// TwinCAT 3 PLC project mobject_motion
// Title: mobject-motion
// Company: mobject-io-ext
// Author: mobject dev team
// ProjectVersion: 0.0.1
// ProgramVersion: 3.1.4023.0
// libraries:
//   mobject-core, * (mobject.io)
//   Tc2_MC2, * (Beckhoff Automation GmbH)
// project tree:
//   Administrative/ ResetCommand.TcPOU, SetPositionCommand.TcPOU
//   Axis/ Axis.TcPOU, I_Axis.TcIO
//   Base/ AxisCommand.TcPOU, I_AxisCommand.TcIO
//   Homing/ DefaultHomingBuilder.TcPOU, HomingCommand.TcPOU, I_DefaultHomingBuilder.TcIO, I_HomingBuilder.TcIO, I_HomingCommand.TcIO, I_PositioningHomingBuilder.TcIO
//   Moves/ DefaultMoveBuilder.TcPOU, I_JogMoveBuilder.TcIO, I_MoveAbsoluteBuilder.TcIO, I_MoveBuilder.TcIO, I_MoveCommand.TcIO, I_MoveRelativeBuilder.TcIO, MoveAbsoluteCommand.TcPOU, MoveAdditiveCommand.TcPOU, MoveCommand.TcPOU, MoveRelativeCommand.TcPOU, MoveVelocityCommand.TcPOU
//   Stops/ HaltCommand.TcPOU, StopCommand.TcPOU
//   Types/ AxisBufferMode.TcDUT, Direction.TcDUT, EncoderReferenceMode.TcDUT, HomingMode.TcDUT, SetPositionMode.TcDUT

// ---- Types/AxisBufferMode.TcDUT
{attribute 'qualified_only'}
{attribute 'strict'}
TYPE AxisBufferMode :
(
	Aborting := MC_Aborting,
	Buffered := MC_Buffered,
	BlendingLow := MC_BlendingLow,
	BlendingPrevious := MC_BlendingPrevious,
	BlendingNext := MC_BlendingNext,
	BlendingHigh := MC_BlendingHigh
) UINT;
END_TYPE

// ---- Types/Direction.TcDUT
{attribute 'qualified_only'}
{attribute 'strict'}
TYPE Direction :
(
    Position := MC_Positive_Direction,
    ShortestWay := MC_Shortest_Way ,
    Negative := MC_Negative_Direction,
    Current := MC_Current_Direction,
	Undefined := MC_Undefined_Direction
) INT;
END_TYPE

// ---- Types/EncoderReferenceMode.TcDUT
// https://infosys.beckhoff.com/english.php?content=../content/1033/ax5000_system_doku_hw2/649689099.html&id=
{attribute 'qualified_only'}
{attribute 'strict'}
TYPE EncoderReferenceMode :
(
	Default := ENCODERREFERENCEMODE_DEFAULT,
	PLCCam := ENCODERREFERENCEMODE_PLCCAM,
	HardwareSync := ENCODERREFERENCEMODE_HARDWARESYNC,
	HardwareLatchPositive := ENCODERREFERENCEMODE_HARDWARELATCHPOS,
	HardwareLatchNegative := ENCODERREFERENCEMODE_HARDWARELATCHNEG,
	SoftwareSync := ENCODERREFERENCEMODE_SOFTWARESYNC,
	SoftwareLatchPositive := ENCODERREFERENCEMODE_SOFTDRIVELATCHPOS,
	SoftwareLatchNegative := ENCODERREFERENCEMODE_SOFTDRIVELATCHNEG
) UDINT;
END_TYPE

// ---- Types/HomingMode.TcDUT
{attribute 'qualified_only'}
{attribute 'strict'}
TYPE HomingMode :
(
	Default := MC_DefaultHoming,
	Direct := MC_Direct,
	ForceCalibration := MC_ForceCalibration,
	ResetCalibration := MC_ResetCalibration
) INT;
END_TYPE

// ---- Types/SetPositionMode.TcDUT
{attribute 'qualified_only'}
{attribute 'strict'}
TYPE SetPositionMode :
(
	Absolute,
	Relative
);
END_TYPE

// ---- Axis/I_Axis.TcIO
INTERFACE I_Axis

PROPERTY INTERNAL _InternalAxisRef : REFERENCE TO Tc2_MC2.AXIS_REF
GET
END_GET
END_PROPERTY

PROPERTY INTERNAL _InternalJog : REFERENCE TO MC_Jog
GET
END_GET
END_PROPERTY

PROPERTY INTERNAL _InternalParameterSet : REFERENCE TO ST_AxisParameterSet
GET
END_GET
END_PROPERTY

PROPERTY AxisId : UDINT
GET
END_GET
END_PROPERTY

{warning 'add property implementation'}
PROPERTY BufferMode : Tc2_MC2.MC_BufferMode
GET
END_GET
SET
END_SET
END_PROPERTY

PROPERTY Busy : BOOL
GET
END_GET
END_PROPERTY

METHOD Disable
END_METHOD

METHOD DisableNegative
END_METHOD

METHOD DisablePositive
END_METHOD

METHOD Enable
VAR_INPUT
	bufferMode : AxisBufferMode;
END_VAR
END_METHOD

METHOD EnableNegative : BOOL
END_METHOD

METHOD EnablePositive
END_METHOD

PROPERTY ErrorId : UDINT
GET
END_GET
END_PROPERTY

METHOD Halt
VAR_INPUT
	feedback : REFERENCE TO I_CommandFeedback;
END_VAR
END_METHOD

PROPERTY HasError : BOOL
GET
END_GET
END_PROPERTY

METHOD HomingBuilder : I_HomingBuilder
END_METHOD

PROPERTY IsAccelerating : BOOL
GET
END_GET
END_PROPERTY

PROPERTY IsAtConstantVelocity : BOOL
GET
END_GET
END_PROPERTY

PROPERTY IsAtStandStill : BOOL
GET
END_GET
END_PROPERTY

PROPERTY IsDecelerating : BOOL
GET
END_GET
END_PROPERTY

PROPERTY IsErrorStopped : BOOL
GET
END_GET
END_PROPERTY

PROPERTY IsHoming : BOOL
GET
END_GET
END_PROPERTY

PROPERTY IsInContinuousMotion : BOOL
GET
END_GET
END_PROPERTY

PROPERTY IsInDiscreteMotion : BOOL
GET
END_GET
END_PROPERTY

PROPERTY IsInSynchronizedMotion : BOOL
GET
END_GET
END_PROPERTY

PROPERTY IsReady : BOOL
GET
END_GET
END_PROPERTY

PROPERTY IsStatusValid : BOOL
GET
END_GET
END_PROPERTY

PROPERTY IsStopping : BOOL
GET
END_GET
END_PROPERTY

METHOD JogBackwards
VAR_INPUT
	velocity : LREAL;
END_VAR
END_METHOD

METHOD JogForward
VAR_INPUT
	velocity : LREAL;
END_VAR
END_METHOD

METHOD MoveBuilder : I_MoveBuilder
END_METHOD

PROPERTY Override : LREAL
GET
END_GET
SET
END_SET
END_PROPERTY

METHOD Reset
VAR_INPUT
	feedback : REFERENCE TO I_CommandFeedback;
END_VAR
END_METHOD

METHOD SetPositionAbsolute
VAR_INPUT
	positionToSet : LREAL;
	feedback : REFERENCE TO I_CommandFeedback;
END_VAR
END_METHOD

METHOD SetPositionRelative
VAR_INPUT
	distanceToShift : LREAL;
	feedback : REFERENCE TO I_CommandFeedback;
END_VAR
END_METHOD

METHOD Stop
VAR_INPUT
	feedback : REFERENCE TO I_CommandFeedback;
END_VAR
END_METHOD

METHOD StopJogging
END_METHOD

END_INTERFACE

// ---- Base/I_AxisCommand.TcIO
INTERFACE I_AxisCommand EXTENDS I_Command

END_INTERFACE

// ---- Homing/I_DefaultHomingBuilder.TcIO
INTERFACE I_DefaultHomingBuilder EXTENDS __System.IQueryInterface

METHOD BuildDefaultHomingCommand : I_HomingCommand
END_METHOD

METHOD Cam : I_DefaultHomingBuilder
VAR_INPUT
	value : REFERENCE TO BOOL;
END_VAR
END_METHOD

METHOD ClearLag : I_PositioningHomingBuilder
END_METHOD

METHOD KeepLag : I_PositioningHomingBuilder
END_METHOD

METHOD Position : I_PositioningHomingBuilder
VAR_INPUT
	value : LREAL;
END_VAR
END_METHOD

METHOD ReferenceMode : I_DefaultHomingBuilder
VAR_INPUT
	value : EncoderReferenceMode;
END_VAR
END_METHOD

METHOD SearchDirection : I_DefaultHomingBuilder
VAR_INPUT
	value : Direction;
END_VAR
END_METHOD

METHOD SearchVelocity : I_DefaultHomingBuilder
VAR_INPUT
	value : LREAL;
END_VAR
END_METHOD

METHOD SyncDirection : I_DefaultHomingBuilder
VAR_INPUT
	value : Direction;
END_VAR
END_METHOD

METHOD SyncVelocity : I_DefaultHomingBuilder
VAR_INPUT
	value : LREAL;
END_VAR
END_METHOD

END_INTERFACE

// ---- Homing/I_HomingBuilder.TcIO
INTERFACE I_HomingBuilder EXTENDS __System.IQueryInterface

METHOD BuildForceCalibrationCommand : I_HomingCommand
END_METHOD

METHOD BuildResetCalibrationCommand : I_HomingCommand
END_METHOD

METHOD Position : I_PositioningHomingBuilder
VAR_INPUT
	value : LREAL;
END_VAR
END_METHOD

END_INTERFACE

// ---- Homing/I_HomingCommand.TcIO
INTERFACE I_HomingCommand EXTENDS I_AxisCommand

END_INTERFACE

// ---- Homing/I_PositioningHomingBuilder.TcIO
INTERFACE I_PositioningHomingBuilder EXTENDS __System.IQueryInterface

METHOD BuildDefaultHomingCommand : I_HomingCommand
END_METHOD

METHOD BuildDirectHomingCommand : I_HomingCommand
END_METHOD

METHOD Cam : I_DefaultHomingBuilder
VAR_INPUT
	value : REFERENCE TO BOOL;
END_VAR
END_METHOD

METHOD ClearLag : I_PositioningHomingBuilder
END_METHOD

METHOD KeepLag : I_PositioningHomingBuilder
END_METHOD

METHOD Position : I_PositioningHomingBuilder
VAR_INPUT
	value : LREAL;
END_VAR
END_METHOD

METHOD ReferenceMode : I_DefaultHomingBuilder
VAR_INPUT
	value : EncoderReferenceMode;
END_VAR
END_METHOD

METHOD SearchDirection : I_DefaultHomingBuilder
VAR_INPUT
	value : Direction;
END_VAR
END_METHOD

METHOD SearchVelocity : I_DefaultHomingBuilder
VAR_INPUT
	value : LREAL;
END_VAR
END_METHOD

METHOD SyncDirection : I_DefaultHomingBuilder
VAR_INPUT
	value : Direction;
END_VAR
END_METHOD

METHOD SyncVelocity : I_DefaultHomingBuilder
VAR_INPUT
	value : LREAL;
END_VAR
END_METHOD

END_INTERFACE

// ---- Moves/I_JogMoveBuilder.TcIO
INTERFACE I_JogMoveBuilder EXTENDS __System.IQueryInterface

METHOD Acceleration : I_MoveBuilder
VAR_INPUT
	value : LREAL;
END_VAR
END_METHOD

METHOD BuildBackwardsCommand : I_MoveCommand
END_METHOD

METHOD BuildForwardCommand : I_MoveCommand
END_METHOD

METHOD Deceleration : I_MoveBuilder
VAR_INPUT
	value : LREAL;
END_VAR
END_METHOD

METHOD Distance : I_JogMoveBuilder
VAR_INPUT
	value : LREAL;
END_VAR
END_METHOD

METHOD Jerk : I_MoveBuilder
VAR_INPUT
	value : LREAL;
END_VAR
END_METHOD

METHOD Velocity : I_MoveBuilder
VAR_INPUT
	value : LREAL;
END_VAR
END_METHOD

END_INTERFACE

// ---- Moves/I_MoveAbsoluteBuilder.TcIO
INTERFACE I_MoveAbsoluteBuilder EXTENDS __System.IQueryInterface

METHOD Acceleration : I_MoveBuilder
VAR_INPUT
	value : LREAL;
END_VAR
END_METHOD

METHOD BufferMode : I_MoveBuilder
VAR_INPUT
	mode : AxisBufferMode;
END_VAR
END_METHOD

METHOD BuildMoveAbsoluteCommand : I_MoveCommand
END_METHOD

METHOD Deceleration : I_MoveBuilder
VAR_INPUT
	value : LREAL;
END_VAR
END_METHOD

METHOD Jerk : I_MoveBuilder
VAR_INPUT
	value : LREAL;
END_VAR
END_METHOD

METHOD Position : I_MoveAbsoluteBuilder
VAR_INPUT
	value : LREAL;
END_VAR
END_METHOD

METHOD Velocity : I_MoveBuilder
VAR_INPUT
	value : LREAL;
END_VAR
END_METHOD

END_INTERFACE

// ---- Moves/I_MoveBuilder.TcIO
INTERFACE I_MoveBuilder EXTENDS __System.IQueryInterface

METHOD Acceleration : I_MoveBuilder
VAR_INPUT
	value : LREAL;
END_VAR
END_METHOD

METHOD BufferMode : I_MoveBuilder
VAR_INPUT
	mode : AxisBufferMode;
END_VAR
END_METHOD

METHOD BuildMoveVelocityCommand : I_MoveCommand
END_METHOD

METHOD Deceleration : I_MoveBuilder
VAR_INPUT
	value : LREAL;
END_VAR
END_METHOD

METHOD Distance : I_MoveRelativeBuilder
VAR_INPUT
	value : LREAL;
END_VAR
END_METHOD

METHOD Jerk : I_MoveBuilder
VAR_INPUT
	value : LREAL;
END_VAR
END_METHOD

METHOD Position : I_MoveAbsoluteBuilder
VAR_INPUT
	value : LREAL;
END_VAR
END_METHOD

METHOD Velocity : I_MoveBuilder
VAR_INPUT
	value : LREAL;
END_VAR
END_METHOD

END_INTERFACE

// ---- Moves/I_MoveCommand.TcIO
INTERFACE I_MoveCommand EXTENDS I_Command

END_INTERFACE

// ---- Moves/I_MoveRelativeBuilder.TcIO
INTERFACE I_MoveRelativeBuilder EXTENDS __System.IQueryInterface

METHOD Acceleration : I_MoveBuilder
VAR_INPUT
	value : LREAL;
END_VAR
END_METHOD

METHOD BufferMode : I_MoveBuilder
VAR_INPUT
	mode : AxisBufferMode;
END_VAR
END_METHOD

METHOD BuildMoveAdditiveCommand : I_MoveCommand
END_METHOD

METHOD BuildMoveRelativeCommand : I_MoveCommand
END_METHOD

METHOD Deceleration : I_MoveBuilder
VAR_INPUT
	value : LREAL;
END_VAR
END_METHOD

METHOD Distance : I_MoveRelativeBuilder
VAR_INPUT
	value : LREAL;
END_VAR
END_METHOD

METHOD Jerk : I_MoveBuilder
VAR_INPUT
	value : LREAL;
END_VAR
END_METHOD

METHOD Velocity : I_MoveBuilder
VAR_INPUT
	value : LREAL;
END_VAR
END_METHOD

END_INTERFACE

// ---- Administrative/ResetCommand.TcPOU
{attribute 'linkalways'} 
{attribute 'no_explicit_call' := 'This FB is a CLASS and must be accessed using methods or properties'}
{attribute 'enable_dynamic_creation'}
FUNCTION_BLOCK ResetCommand EXTENDS AxisCommand

METHOD FB_init : BOOL
VAR_INPUT
	bInitRetains : BOOL; // if TRUE, the retain variables are initialized (warm start / cold start)
	bInCopyCode : BOOL;  // if TRUE, the instance afterwards gets moved into the copy code (online change)
	axis : I_Axis;
END_VAR
_axis := axis;
END_METHOD

METHOD PROTECTED  WhileBusy
VAR_INPUT
	CommandState : I_CommandBusyState;
END_VAR
VAR_INST
	_fb : MC_Reset;
END_VAR
_fb(
	Axis := _axis._InternalAxisRef,
	Execute := TRUE
);

IF _fb.Busy THEN
	RETURN;
END_IF

_fb(Axis := _axis._InternalAxisRef, Execute := FALSE);

IF _fb.Error THEN
	CommandState.SetError(_fb.ErrorID);
	RETURN;
END_IF

CommandState.SetDone();
END_METHOD

END_FUNCTION_BLOCK

// ---- Base/AxisCommand.TcPOU
{attribute 'linkalways'} 
{attribute 'no_explicit_call' := 'This FB is a CLASS and must be accessed using methods or properties'}
{attribute 'enable_dynamic_creation'}
FUNCTION_BLOCK ABSTRACT AxisCommand EXTENDS Command IMPLEMENTS I_AxisCommand
VAR
	_axis : I_Axis;
END_VAR

END_FUNCTION_BLOCK

// ---- Axis/Axis.TcPOU
{attribute 'linkalways'} 
{attribute 'no_explicit_call' := 'This FB is a CLASS and must be accessed using methods or properties'}
{attribute 'enable_dynamic_creation'}
FUNCTION_BLOCK Axis EXTENDS CyclicInstance IMPLEMENTS I_Axis
VAR
	_axisRef : Tc2_MC2.AXIS_REF;
	_power : MC_Power;
	_jog : MC_Jog;
	_readStatus : MC_ReadStatus;
	_parameterSet : ST_AxisParameterSet;
	
	_enable : BOOL;
	_enablePositive : BOOL;
	_enableNegative : BOOL;
	
	_override : LREAL := 100.0;
	_powerBufferMode : AxisBufferMode := AxisBufferMode.Aborting;
END_VAR

PROPERTY PUBLIC _InternalAxisRef : REFERENCE TO Tc2_MC2.AXIS_REF
GET
_InternalAxisRef REF= _axisRef;
END_GET
END_PROPERTY

PROPERTY PUBLIC _InternalJog : REFERENCE TO MC_Jog
GET
_InternalJog REF= _jog;
END_GET
END_PROPERTY

PROPERTY PUBLIC _InternalParameterSet : REFERENCE TO ST_AxisParameterSet
GET
_InternalParameterSet REF= _parameterSet;
END_GET
END_PROPERTY

PROPERTY AxisId : UDINT
GET
AxisId := _axisRef.NcToPlc.AxisId;
END_GET
END_PROPERTY

{warning 'add property implementation'}
PROPERTY BufferMode : Tc2_MC2.MC_BufferMode
GET
END_GET
SET
END_SET
END_PROPERTY

PROPERTY Busy : BOOL
GET
END_GET
END_PROPERTY

METHOD  CyclicCall
VAR_INST
	_readParameterSet : MC_ReadParameterSet;
	parameterSetRead : BOOL;
END_VAR
_power(
	Axis := THIS^._axisRef,
	Enable := THIS^._enable,
	Enable_Positive := THIS^._enablePositive,
	Enable_Negative := THIS^._enableNegative,
	Override := THIS^._override,
	BufferMode := THIS^._powerBufferMode
);

_readStatus(
	Axis := THIS^._axisRef,
	Enable := _enable
);

IF NOT parameterSetRead THEN
	_readParameterSet(
		Axis := THIS^._axisRef,
		Parameter := _parameterSet,
		Execute := TRUE
	);
	
	IF NOT _readParameterSet.Busy THEN
		_readParameterSet(
			Axis := THIS^._axisRef,
			Parameter := _parameterSet,
			Execute := TRUE
		);
		IF _readParameterSet.Done THEN
			parameterSetRead := TRUE;
		END_IF
	END_IF
END_IF
END_METHOD

METHOD Disable
_enable := FALSE;
END_METHOD

METHOD DisableNegative
_enableNegative := FALSE;
END_METHOD

METHOD DisablePositive
_enablePositive := FALSE;
END_METHOD

METHOD Enable
VAR_INPUT
	bufferMode : AxisBufferMode;
END_VAR
_enable := TRUE;
_powerBufferMode := bufferMode;
END_METHOD

METHOD EnableNegative : BOOL
_enableNegative := TRUE;
END_METHOD

METHOD EnablePositive
_enablePositive := TRUE;
END_METHOD

PROPERTY ErrorId : UDINT
GET
ErrorId := _readStatus.ErrorID;
END_GET
END_PROPERTY

METHOD Halt
VAR_INPUT
	feedback : REFERENCE TO I_CommandFeedback;
END_VAR
VAR_INST
	pCmd : POINTER TO HaltCommand;
END_VAR
pCmd := __NEW(HaltCommand(axis := THIS^));
pCmd^.Execute(feedback).ThenRelease();
END_METHOD

PROPERTY HasError : BOOL
GET
HasError := _readStatus.Error;
END_GET
END_PROPERTY

METHOD HomingBuilder : I_HomingBuilder
VAR_INST
	builder : DefaultHomingBuilder(axis := THIS^);
END_VAR
HomingBuilder := builder;
END_METHOD

PROPERTY IsAccelerating : BOOL
GET
IsAccelerating := _readStatus.Accelerating;
END_GET
END_PROPERTY

PROPERTY IsAtConstantVelocity : BOOL
GET
IsAtConstantVelocity := _readStatus.ConstantVelocity;
END_GET
END_PROPERTY

PROPERTY IsAtStandStill : BOOL
GET
IsAtStandStill := _readStatus.StandStill;
END_GET
END_PROPERTY

PROPERTY IsDecelerating : BOOL
GET
IsDecelerating := _readStatus.Decelerating;
END_GET
END_PROPERTY

PROPERTY IsErrorStopped : BOOL
GET
IsErrorStopped := _readStatus.ErrorStop;
END_GET
END_PROPERTY

PROPERTY IsHoming : BOOL
GET
IsHoming := _readStatus.Homing;
END_GET
END_PROPERTY

PROPERTY IsInContinuousMotion : BOOL
GET
IsInContinuousMotion := _readStatus.ContinuousMotion;
END_GET
END_PROPERTY

PROPERTY IsInDiscreteMotion : BOOL
GET
IsInDiscreteMotion := _readStatus.DiscreteMotion;
END_GET
END_PROPERTY

PROPERTY IsInSynchronizedMotion : BOOL
GET
IsInSynchronizedMotion := _readStatus.SynchronizedMotion;
END_GET
END_PROPERTY

PROPERTY IsReady : BOOL
GET
IsReady := _power.Status;
END_GET
END_PROPERTY

PROPERTY IsStatusValid : BOOL
GET
IsStatusValid := _readStatus.Valid;
END_GET
END_PROPERTY

PROPERTY IsStopping : BOOL
GET
IsStopping := _readStatus.Stopping;
END_GET
END_PROPERTY

METHOD JogBackwards
VAR_INPUT
	velocity : LREAL;
END_VAR
_jog(
	Axis := _axisRef,
	JogForward := FALSE,
	JogBackwards := TRUE,
	Mode := MC_JOGMODE_CONTINOUS,
	Velocity := velocity
);
END_METHOD

METHOD JogForward
VAR_INPUT
	velocity : LREAL;
END_VAR
_jog(
	Axis := _axisRef,
	JogForward := TRUE,
	JogBackwards := FALSE,
	Mode := MC_JOGMODE_CONTINOUS,
	Velocity := velocity
);
END_METHOD

METHOD MoveBuilder : I_MoveBuilder
VAR_INST
	builder : DefaultMoveBuilder(axis := THIS^);
END_VAR
MoveBuilder := builder;
END_METHOD

PROPERTY Override : LREAL
GET
Override := _override;
END_GET
SET
_override := Override;
END_SET
END_PROPERTY

METHOD Reset
VAR_INPUT
	feedback : REFERENCE TO I_CommandFeedback;
END_VAR
VAR_INST
	pCmd : POINTER TO ResetCommand;
END_VAR
pCmd := __NEW(ResetCommand(axis := THIS^));
pCmd^.Execute(feedback).ThenRelease();
END_METHOD

METHOD SetPositionAbsolute
VAR_INPUT
	positionToSet : LREAL;
	feedback : REFERENCE TO I_CommandFeedback;
END_VAR
VAR_INST
	pCmd : POINTER TO SetPositionCommand;
END_VAR
pCmd := __NEW(SetPositionCommand(axis := THIS^, position := positionToSet, mode := SetPositionMode.Absolute));
pCmd^.Execute(feedback).ThenRelease();
END_METHOD

METHOD SetPositionRelative
VAR_INPUT
	distanceToShift : LREAL;
	feedback : REFERENCE TO I_CommandFeedback;
END_VAR
VAR_INST
	pCmd : POINTER TO SetPositionCommand;
END_VAR
pCmd := __NEW(SetPositionCommand(axis := THIS^, position := distanceToShift, mode := SetPositionMode.Relative));
pCmd^.Execute(feedback).ThenRelease();
END_METHOD

METHOD Stop
VAR_INPUT
	feedback : REFERENCE TO I_CommandFeedback;
END_VAR
VAR_INST
	pCmd : POINTER TO StopCommand;
END_VAR
pCmd := __NEW(StopCommand(axis := THIS^));
pCmd^.Execute(feedback).ThenRelease();
END_METHOD

METHOD StopJogging
_jog(
	Axis := _axisRef,
	JogForward := FALSE,
	JogBackwards := FALSE,
);
END_METHOD

END_FUNCTION_BLOCK

// ---- Stops/HaltCommand.TcPOU
{attribute 'linkalways'} 
{attribute 'no_explicit_call' := 'This FB is a CLASS and must be accessed using methods or properties'}
{attribute 'enable_dynamic_creation'}
FUNCTION_BLOCK HaltCommand EXTENDS AxisCommand
VAR
	_deceleration : LREAL;
	_jerk : LREAL;
	_bufferMode : AxisBufferMode;
END_VAR

METHOD FB_init : BOOL
VAR_INPUT
	bInitRetains : BOOL; // if TRUE, the retain variables are initialized (warm start / cold start)
	bInCopyCode : BOOL;  // if TRUE, the instance afterwards gets moved into the copy code (online change)
	axis : I_Axis;
END_VAR
_axis := axis;
END_METHOD

METHOD PROTECTED  WhileBusy
VAR_INPUT
	CommandState : I_CommandBusyState;
END_VAR
VAR_INST
	_fb : MC_Halt;
END_VAR
_fb(
	Axis := _axis._InternalAxisRef,
	Execute := TRUE,
	Deceleration := _deceleration,
	Jerk := _jerk,
	BufferMode := _bufferMode
);

IF _fb.Busy THEN
	RETURN;
END_IF

_fb(Axis := _axis._InternalAxisRef, Execute := FALSE);

IF _fb.CommandAborted THEN
	CommandState.SetAborting();
	RETURN;
END_IF

IF _fb.Error THEN
	CommandState.SetError(_fb.ErrorID);
	RETURN;
END_IF

CommandState.SetDone();
END_METHOD

END_FUNCTION_BLOCK

// ---- Homing/DefaultHomingBuilder.TcPOU
{attribute 'linkalways'} 
{attribute 'no_explicit_call' := 'This FB is a CLASS and must be accessed using methods or properties'}
{attribute 'enable_dynamic_creation'}
FUNCTION_BLOCK DefaultHomingBuilder IMPLEMENTS I_HomingBuilder, I_PositioningHomingBuilder, I_DefaultHomingBuilder
VAR
	_axis : I_Axis;
	_position : LREAL;
	_options : ST_HomingOptions;
	_cam : REFERENCE TO BOOL;
END_VAR

METHOD BuildDefaultHomingCommand : I_HomingCommand
VAR
	pCmd : POINTER TO HomingCommand;
	cmd : I_HomingCommand;
END_VAR
pCmd := __NEW(HomingCommand(
	axis := _axis,
	position := _position,
	mode := HomingMode.Default,
	options := _options,
	cam := _cam
));
BuildDefaultHomingCommand := pCmd^;
END_METHOD

METHOD BuildDirectHomingCommand : I_HomingCommand
VAR
	pCmd : POINTER TO HomingCommand;
	cmd : I_HomingCommand;
	null : BOOL;
END_VAR
pCmd := __NEW(HomingCommand(
	axis := _axis,
	position := _position,
	mode := HomingMode.Direct,
	options := _options,
	cam := null
));
BuildDirectHomingCommand := pCmd^;
END_METHOD

METHOD BuildForceCalibrationCommand : I_HomingCommand
VAR
	pCmd : POINTER TO HomingCommand;
	cmd : I_HomingCommand;
	null : BOOL;
END_VAR
pCmd := __NEW(HomingCommand(
	axis := _axis,
	position := _position,
	mode := HomingMode.ForceCalibration,
	options := _options,
	cam := null
));
BuildForceCalibrationCommand := pCmd^;
END_METHOD

METHOD BuildResetCalibrationCommand : I_HomingCommand
VAR
	pCmd : POINTER TO HomingCommand;
	cmd : I_HomingCommand;
	null : BOOL;
END_VAR
pCmd := __NEW(HomingCommand(
	axis := _axis,
	position := _position,
	mode := HomingMode.ResetCalibration,
	options := _options,
	cam := null
));
BuildResetCalibrationCommand := pCmd^;
END_METHOD

METHOD Cam : I_DefaultHomingBuilder
VAR_INPUT
	value : REFERENCE TO BOOL;
END_VAR
_cam REF= value;
Cam := THIS^;
END_METHOD

METHOD ClearLag : I_PositioningHomingBuilder
_options.ClearPositionLag := TRUE;
ClearLag := THIS^;
END_METHOD

METHOD FB_init : BOOL
VAR_INPUT
	bInitRetains : BOOL; // if TRUE, the retain variables are initialized (warm start / cold start)
	bInCopyCode : BOOL;  // if TRUE, the instance afterwards gets moved into the copy code (online change)
	axis : I_Axis;
END_VAR
_axis := axis;
END_METHOD

METHOD KeepLag : I_PositioningHomingBuilder
_options.ClearPositionLag := FALSE;
KeepLag := THIS^;
END_METHOD

METHOD Position : I_PositioningHomingBuilder
VAR_INPUT
	value : LREAL;
END_VAR
_position := value;
Position := THIS^;
END_METHOD

METHOD ReferenceMode : I_DefaultHomingBuilder
VAR_INPUT
	value : EncoderReferenceMode;
END_VAR
_options.ReferenceMode := value;
ReferenceMode := THIS^;
END_METHOD

METHOD SearchDirection : I_DefaultHomingBuilder
VAR_INPUT
	value : Direction;
END_VAR
_options.SearchDirection := value;
SearchDirection := THIS^;
END_METHOD

METHOD SearchVelocity : I_DefaultHomingBuilder
VAR_INPUT
	value	: LREAL;
END_VAR
_options.SearchVelocity := value;
SearchVelocity := THIS^;
END_METHOD

METHOD SyncDirection : I_DefaultHomingBuilder
VAR_INPUT
	value : Direction;
END_VAR
_options.SyncDirection := value;
SyncDirection := THIS^;
END_METHOD

METHOD SyncVelocity : I_DefaultHomingBuilder
VAR_INPUT
	value : LREAL;
END_VAR
_options.SyncVelocity := value;
SyncVelocity := THIS^;
END_METHOD

END_FUNCTION_BLOCK

// ---- Homing/HomingCommand.TcPOU
{attribute 'linkalways'} 
{attribute 'no_explicit_call' := 'This FB is a CLASS and must be accessed using methods or properties'}
{attribute 'enable_dynamic_creation'}
FUNCTION_BLOCK HomingCommand EXTENDS AxisCommand IMPLEMENTS I_HomingCommand
VAR
	_fb : MC_Home;
	_position : LREAL;
	_mode : HomingMode;
	_options : ST_HomingOptions;
	_cam : REFERENCE TO BOOL;
END_VAR

METHOD FB_init : BOOL
VAR_INPUT
	bInitRetains : BOOL; // if TRUE, the retain variables are initialized (warm start / cold start)
	bInCopyCode : BOOL;  // if TRUE, the instance afterwards gets moved into the copy code (online change)
	axis : I_Axis;
	position : LREAL;
	mode : HomingMode;
	options : ST_HomingOptions;
	cam : REFERENCE TO BOOL;
END_VAR
_axis := axis;
_position := position;
_mode := mode;
_options := options;
IF __ISVALIDREF(cam) THEN
	_cam REF= cam;
END_IF
END_METHOD

METHOD PROTECTED  WhileBusy
VAR_INPUT
	CommandState : I_CommandBusyState;
END_VAR
VAR
	_dummy : BOOL := FALSE;
END_VAR
VAR_INST
	_fb : MC_Home;
END_VAR
IF NOT __ISVALIDREF(_cam) THEN
	_cam REF= _dummy;
END_IF

_fb(
	Axis := _axis._InternalAxisRef,
	Execute := TRUE,
	Position := _position,
	HomingMode := _mode,
	Options := _options,
	bCalibrationCam := _cam
);

IF _fb.Busy THEN
	RETURN;
END_IF

IF _fb.CommandAborted THEN
	_fb(Axis := _axis._InternalAxisRef, Execute := FALSE);
	CommandState.SetAborting();
	RETURN;
END_IF

IF _fb.Error THEN
	_fb(Axis := _axis._InternalAxisRef, Execute := FALSE);
	CommandState.SetError(_fb.ErrorID);
	RETURN;
END_IF

_fb(Axis := _axis._InternalAxisRef, Execute := FALSE);
CommandState.SetDone();
END_METHOD

END_FUNCTION_BLOCK

// ---- Moves/DefaultMoveBuilder.TcPOU
{attribute 'linkalways'} 
{attribute 'no_explicit_call' := 'This FB is a CLASS and must be accessed using methods or properties'}
{attribute 'enable_dynamic_creation'}
FUNCTION_BLOCK DefaultMoveBuilder IMPLEMENTS I_MoveBuilder, I_MoveAbsoluteBuilder, I_MoveRelativeBuilder
VAR
	_axis : I_Axis;
	_position : LREAL;
	_distance : LREAL;
	_velocity : LREAL;
	_acceleration: LREAL;
	_deceleration: LREAL;
	_jerk: LREAL;
	_bufferMode: AxisBufferMode;
END_VAR

METHOD Acceleration : I_MoveBuilder
VAR_INPUT
	value : LREAL;
END_VAR
_acceleration := value;
Acceleration := THIS^;
END_METHOD

METHOD BufferMode : I_MoveBuilder
VAR_INPUT
	mode : AxisBufferMode;
END_VAR
_bufferMode := mode;
BufferMode := THIS^;
END_METHOD

METHOD BuildMoveAbsoluteCommand : I_MoveCommand
VAR
	pCmd : POINTER TO MoveAbsoluteCommand;
	cmd : I_MoveCommand;
END_VAR
pCmd := __NEW(MoveAbsoluteCommand(
	axis := _axis,
	position := _position,
	velocity := _velocity,
	acceleration := _acceleration,
	deceleration := _deceleration,
	jerk := _jerk,
	bufferMode := _bufferMode
));
BuildMoveAbsoluteCommand := pCmd^;
END_METHOD

METHOD BuildMoveAdditiveCommand : I_MoveCommand
VAR
	pCmd : POINTER TO MoveAdditiveCommand;
	cmd : I_MoveCommand;
END_VAR
pCmd := __NEW(MoveAdditiveCommand(
	axis := _axis,
	distance := _distance,
	velocity := _velocity,
	acceleration := _acceleration,
	deceleration := _deceleration,
	jerk := _jerk,
	bufferMode := _bufferMode
));
BuildMoveAdditiveCommand := pCmd^;
END_METHOD

METHOD BuildMoveRelativeCommand : I_MoveCommand
VAR
	pCmd : POINTER TO MoveRelativeCommand;
	cmd : I_MoveCommand;
END_VAR
pCmd := __NEW(MoveRelativeCommand(
	axis := _axis,
	distance := _distance,
	velocity := _velocity,
	acceleration := _acceleration,
	deceleration := _deceleration,
	jerk := _jerk,
	bufferMode := _bufferMode
));
BuildMoveRelativeCommand := pCmd^;
END_METHOD

METHOD BuildMoveVelocityCommand : I_MoveCommand
VAR
	pCmd : POINTER TO MoveVelocityCommand;
	cmd : I_MoveCommand;
END_VAR
pCmd := __NEW(MoveVelocityCommand(
	axis := _axis,
	velocity := _velocity,
	acceleration := _acceleration,
	deceleration := _deceleration,
	jerk := _jerk,
	bufferMode := _bufferMode
));
BuildMoveVelocityCommand := pCmd^;
END_METHOD

METHOD Deceleration : I_MoveBuilder
VAR_INPUT
	value : LREAL;
END_VAR
_deceleration := value;
Deceleration := THIS^;
END_METHOD

METHOD Distance : I_MoveRelativeBuilder
VAR_INPUT
	value : LREAL;
END_VAR
_distance := value;
Distance := THIS^;
END_METHOD

METHOD FB_init : BOOL
VAR_INPUT
	bInitRetains : BOOL; // if TRUE, the retain variables are initialized (warm start / cold start)
	bInCopyCode : BOOL;  // if TRUE, the instance afterwards gets moved into the copy code (online change)
	axis : I_Axis;
END_VAR
_axis := axis;
END_METHOD

METHOD Jerk : I_MoveBuilder
VAR_INPUT
	value : LREAL;
END_VAR
_jerk := value;
Jerk := THIS^;
END_METHOD

METHOD Position : I_MoveAbsoluteBuilder
VAR_INPUT
	value : LREAL;
END_VAR
_position := value;
Position := THIS^;
END_METHOD

METHOD Velocity : I_MoveBuilder
VAR_INPUT
	value : LREAL;
END_VAR
IF value <= 0 THEN
	_velocity := _axis._InternalParameterSet.fDriveVeloReferenz;
ELSE
	_velocity := value;
END_IF
Velocity := THIS^;
END_METHOD

END_FUNCTION_BLOCK

// ---- Moves/MoveAbsoluteCommand.TcPOU
{attribute 'linkalways'} 
{attribute 'no_explicit_call' := 'This FB is a CLASS and must be accessed using methods or properties'}
{attribute 'enable_dynamic_creation'}
FUNCTION_BLOCK INTERNAL MoveAbsoluteCommand EXTENDS MoveCommand
VAR
	_fb : MC_MoveAbsolute;
	_position : LREAL;
END_VAR

METHOD FB_init : BOOL
VAR_INPUT
	bInitRetains : BOOL; // if TRUE, the retain variables are initialized (warm start / cold start)
	bInCopyCode : BOOL;  // if TRUE, the instance afterwards gets moved into the copy code (online change)
	axis : I_Axis;
	position : LREAL;
	velocity : LREAL;
	acceleration : LREAL;
	deceleration : LREAL;
	jerk : LREAL;
	bufferMode : AxisBufferMode;
END_VAR
_axis := axis;
_position := position;
_velocity := velocity;
_acceleration := acceleration;
_deceleration := deceleration;
_jerk := jerk;
_bufferMode := bufferMode;
END_METHOD

METHOD PROTECTED WhileBusy
VAR_INPUT
	CommandState : I_CommandBusyState;
END_VAR
_fb(
	Axis := _axis._InternalAxisRef,
	Execute := TRUE,
	Position := _position,
	Velocity := _velocity,
	Acceleration := _acceleration,
	Deceleration := _deceleration,
	Jerk := _jerk,
	BufferMode := _bufferMode
);

IF _fb.Busy THEN
	RETURN;
END_IF

IF _fb.CommandAborted THEN
	_fb(Axis := _axis._InternalAxisRef, Execute := FALSE);
	CommandState.SetAborting();
	RETURN;
END_IF

IF _fb.Error THEN
	_fb(Axis := _axis._InternalAxisRef, Execute := FALSE);
	CommandState.SetError(_fb.ErrorID);
	RETURN;
END_IF

_fb(Axis := _axis._InternalAxisRef, Execute := FALSE);
CommandState.SetDone();
END_METHOD

END_FUNCTION_BLOCK

// ---- Moves/MoveCommand.TcPOU
{attribute 'linkalways'} 
{attribute 'no_explicit_call' := 'This FB is a CLASS and must be accessed using methods or properties'}
{attribute 'enable_dynamic_creation'}
FUNCTION_BLOCK ABSTRACT MoveCommand EXTENDS AxisCommand IMPLEMENTS I_MoveCommand
VAR
	_velocity : LREAL;
	_acceleration: LREAL;
	_deceleration: LREAL;
	_jerk: LREAL;
	_bufferMode: AxisBufferMode;
END_VAR

END_FUNCTION_BLOCK

// ---- Moves/MoveAdditiveCommand.TcPOU
{attribute 'linkalways'} 
{attribute 'no_explicit_call' := 'This FB is a CLASS and must be accessed using methods or properties'}
{attribute 'enable_dynamic_creation'}
FUNCTION_BLOCK INTERNAL MoveAdditiveCommand EXTENDS MoveCommand
VAR
	_fb : MC_MoveAdditive;
	_distance : LREAL;
END_VAR

METHOD FB_init : BOOL
VAR_INPUT
	bInitRetains : BOOL; // if TRUE, the retain variables are initialized (warm start / cold start)
	bInCopyCode : BOOL;  // if TRUE, the instance afterwards gets moved into the copy code (online change)
	axis : I_Axis;
	distance : LREAL;
	velocity : LREAL;
	acceleration : LREAL;
	deceleration : LREAL;
	jerk : LREAL;
	bufferMode : AxisBufferMode;
END_VAR
_axis := axis;
_distance := distance;
_velocity := velocity;
_acceleration := acceleration;
_deceleration := deceleration;
_jerk := jerk;
_bufferMode := bufferMode;
END_METHOD

METHOD PROTECTED WhileBusy
VAR_INPUT
	CommandState : I_CommandBusyState;
END_VAR
_fb(
	Axis := _axis._InternalAxisRef,
	Execute := TRUE,
	Distance := _distance,
	Velocity := _velocity,
	Acceleration := _acceleration,
	Deceleration := _deceleration,
	Jerk := _jerk,
	BufferMode := _bufferMode
);

IF _fb.Busy THEN
	RETURN;
END_IF

IF _fb.CommandAborted THEN
	_fb(Axis := _axis._InternalAxisRef, Execute := FALSE);
	CommandState.SetAborting();
	RETURN;
END_IF

IF _fb.Error THEN
	_fb(Axis := _axis._InternalAxisRef, Execute := FALSE);
	CommandState.SetError(_fb.ErrorID);
	RETURN;
END_IF

_fb(Axis := _axis._InternalAxisRef, Execute := FALSE);
CommandState.SetDone();
END_METHOD

END_FUNCTION_BLOCK

// ---- Moves/MoveRelativeCommand.TcPOU
{attribute 'linkalways'} 
{attribute 'no_explicit_call' := 'This FB is a CLASS and must be accessed using methods or properties'}
{attribute 'enable_dynamic_creation'}
FUNCTION_BLOCK INTERNAL MoveRelativeCommand EXTENDS MoveCommand
VAR
	_fb : MC_MoveRelative;
	_distance : LREAL;
END_VAR

METHOD FB_init : BOOL
VAR_INPUT
	bInitRetains : BOOL; // if TRUE, the retain variables are initialized (warm start / cold start)
	bInCopyCode : BOOL;  // if TRUE, the instance afterwards gets moved into the copy code (online change)
	axis : I_Axis;
	distance : LREAL;
	velocity : LREAL;
	acceleration : LREAL;
	deceleration : LREAL;
	jerk : LREAL;
	bufferMode : AxisBufferMode;
END_VAR
_axis := axis;
_distance := distance;
_velocity := velocity;
_acceleration := acceleration;
_deceleration := deceleration;
_jerk := jerk;
_bufferMode := bufferMode;
END_METHOD

METHOD PROTECTED WhileBusy
VAR_INPUT
	CommandState : I_CommandBusyState;
END_VAR
_fb(
	Axis := _axis._InternalAxisRef,
	Execute := TRUE,
	Distance := _distance,
	Velocity := _velocity,
	Acceleration := _acceleration,
	Deceleration := _deceleration,
	Jerk := _jerk,
	BufferMode := _bufferMode
);

IF _fb.Busy THEN
	RETURN;
END_IF

IF _fb.CommandAborted THEN
	_fb(Axis := _axis._InternalAxisRef, Execute := FALSE);
	CommandState.SetAborting();
	RETURN;
END_IF

IF _fb.Error THEN
	_fb(Axis := _axis._InternalAxisRef, Execute := FALSE);
	CommandState.SetError(_fb.ErrorID);
	RETURN;
END_IF

_fb(Axis := _axis._InternalAxisRef, Execute := FALSE);
CommandState.SetDone();
END_METHOD

END_FUNCTION_BLOCK

// ---- Moves/MoveVelocityCommand.TcPOU
{attribute 'linkalways'} 
{attribute 'no_explicit_call' := 'This FB is a CLASS and must be accessed using methods or properties'}
{attribute 'enable_dynamic_creation'}
FUNCTION_BLOCK INTERNAL MoveVelocityCommand EXTENDS MoveCommand
VAR
	_fb : MC_MoveVelocity;
END_VAR

METHOD FB_init : BOOL
VAR_INPUT
	bInitRetains : BOOL; // if TRUE, the retain variables are initialized (warm start / cold start)
	bInCopyCode : BOOL;  // if TRUE, the instance afterwards gets moved into the copy code (online change)
	axis : I_Axis;
	velocity : LREAL;
	acceleration : LREAL;
	deceleration : LREAL;
	jerk : LREAL;
	bufferMode : AxisBufferMode;
END_VAR
_axis := axis;
_velocity := velocity;
_acceleration := acceleration;
_deceleration := deceleration;
_jerk := jerk;
_bufferMode := bufferMode;
END_METHOD

METHOD PROTECTED WhileBusy
VAR_INPUT
	CommandState : I_CommandBusyState;
END_VAR
_fb(
	Axis := _axis._InternalAxisRef,
	Execute := TRUE,
	Velocity := _velocity,
	Acceleration := _acceleration,
	Deceleration := _deceleration,
	Jerk := _jerk,
	BufferMode := _bufferMode
);

IF _fb.Busy THEN
	RETURN;
END_IF

IF _fb.CommandAborted THEN
	_fb(Axis := _axis._InternalAxisRef, Execute := FALSE);
	CommandState.SetAborting();
	RETURN;
END_IF

IF _fb.Error THEN
	_fb(Axis := _axis._InternalAxisRef, Execute := FALSE);
	CommandState.SetError(_fb.ErrorID);
	RETURN;
END_IF

_fb(Axis := _axis._InternalAxisRef, Execute := FALSE);
CommandState.SetDone();
END_METHOD

END_FUNCTION_BLOCK

// ---- Administrative/SetPositionCommand.TcPOU
{attribute 'linkalways'} 
{attribute 'no_explicit_call' := 'This FB is a CLASS and must be accessed using methods or properties'}
{attribute 'enable_dynamic_creation'}
FUNCTION_BLOCK SetPositionCommand EXTENDS AxisCommand
VAR
	_position : LREAL;
	_mode : SetPositionMode;
END_VAR

METHOD FB_init : BOOL
VAR_INPUT
	bInitRetains : BOOL; // if TRUE, the retain variables are initialized (warm start / cold start)
	bInCopyCode : BOOL;  // if TRUE, the instance afterwards gets moved into the copy code (online change)
	axis : I_Axis;
	position : LREAL;
	mode : SetPositionMode;
END_VAR
_axis := axis;
_position := position;
_mode := mode;
END_METHOD

METHOD PROTECTED  WhileBusy
VAR_INPUT
	CommandState : I_CommandBusyState;
END_VAR
VAR_INST
	_fb : MC_SetPosition;
END_VAR
_fb(
	Axis := _axis._InternalAxisRef,
	Execute := TRUE,
	Position := _position,
	Mode := (_mode = SetPositionMode.Relative)
);

IF _fb.Busy THEN
	RETURN;
END_IF

_fb(Axis := _axis._InternalAxisRef, Execute := FALSE);

IF _fb.Error THEN
	CommandState.SetError(_fb.ErrorID);
	RETURN;
END_IF

CommandState.SetDone();
END_METHOD

END_FUNCTION_BLOCK

// ---- Stops/StopCommand.TcPOU
{attribute 'linkalways'} 
{attribute 'no_explicit_call' := 'This FB is a CLASS and must be accessed using methods or properties'}
{attribute 'enable_dynamic_creation'}
FUNCTION_BLOCK StopCommand EXTENDS AxisCommand
VAR
	_deceleration : LREAL;
	_jerk : LREAL;
END_VAR

METHOD FB_init : BOOL
VAR_INPUT
	bInitRetains : BOOL; // if TRUE, the retain variables are initialized (warm start / cold start)
	bInCopyCode : BOOL;  // if TRUE, the instance afterwards gets moved into the copy code (online change)
	axis : I_Axis;
END_VAR
_axis := axis;
END_METHOD

METHOD PROTECTED WhileBusy
VAR_INPUT
	CommandState : I_CommandBusyState;
END_VAR
VAR_INST
	_fb : MC_Stop;
END_VAR
_fb(
	Axis := _axis._InternalAxisRef,
	Execute := TRUE,
	Deceleration := _deceleration,
	Jerk := _jerk
);

IF NOT _fb.Done THEN
	RETURN;
END_IF

_fb(Axis := _axis._InternalAxisRef, Execute := FALSE);
CommandState.SetDone();
END_METHOD

END_FUNCTION_BLOCK
